{attribute 'GeneratedUsingTerminal: EK1100-0000-0018'}
{attribute addProperty BoxType "EK1100-0000-0018"}
{attribute addProperty Id "Beckhoff_ELM37xxEK1122Beckhoff_ELM37xxEK1122_E40DDF852A_0001_ELM3702_0000_0016ELM3702_B416BFEF50A_0002_ELM3702_0000_0017ELM3702_B416BFEF50A_0003_ELM3704_0000_0016ELM3704_9E251EA472A_0004_ELM3704_0000_0017ELM3704_9E251EA472A_0005_ELM3704_0001_0017ELM3704_9E251EA472A_0006_ELM3704_0020_0016ELM3704_9E251EA472A_0007_ELM3702_0101_0016ELM3702_B416BFEF50A_0008_ELM3704_1001_0016ELM3704_9E251EA472A_0009_ELM3704_1001_0017ELM3704_9E251EA472"}
{attribute addProperty CRC "1942405192"}
{attribute addProperty Size "584"}
TYPE Beckhoff_ELM37xx_73C6C048 EXTENDS EK1100_1FC0878B :
STRUCT
	{attribute addProperty Name "Beckhoff_ELM37xxEK1122"}
	Beckhoff_ELM37xxEK1122 : Beckhoff_ELM37xxEK1122_E40DDF85;
	{attribute addProperty Name "A_0001_ELM3702_0000_0016"}
	A_0001_ELM3702_0000_0016 : ELM3702_B416BFEF;
	{attribute addProperty Name "A_0002_ELM3702_0000_0017"}
	A_0002_ELM3702_0000_0017 : ELM3702_B416BFEF;
	{attribute addProperty Name "A_0003_ELM3704_0000_0016"}
	A_0003_ELM3704_0000_0016 : ELM3704_9E251EA4;
	{attribute addProperty Name "A_0004_ELM3704_0000_0017"}
	A_0004_ELM3704_0000_0017 : ELM3704_9E251EA4;
	{attribute addProperty Name "A_0005_ELM3704_0001_0017"}
	A_0005_ELM3704_0001_0017 : ELM3704_9E251EA4;
	{attribute addProperty Name "A_0006_ELM3704_0020_0016"}
	A_0006_ELM3704_0020_0016 : ELM3704_9E251EA4;
	{attribute addProperty Name "A_0007_ELM3702_0101_0016"}
	A_0007_ELM3702_0101_0016 : ELM3702_B416BFEF;
	{attribute addProperty Name "A_0008_ELM3704_1001_0016"}
	A_0008_ELM3704_1001_0016 : ELM3704_9E251EA4;
	{attribute addProperty Name "A_0009_ELM3704_1001_0017"}
	A_0009_ELM3704_1001_0017 : ELM3704_9E251EA4;
END_STRUCT
END_TYPE

(* stored: Version 1.2.0.0, ProductVersion 3.1.4024.9
   DUT Beckhoff_ELM37xx_73C6C048: Id {e41eeda7-9d77-4412-a1d3-c2648532a9ca} *)
